// TIA Portal project "SistemaSemaforico_Curto_Claudio" (V15.1)

(* hardware
DEVICE "S7-1200 station_1"  S7-1200 Station
   slot 0: "Telaio di montaggio_0"  S7-1200 Rack  Rack  V1.0
   slot 1: "PLC_1"  CPU 1214C DC/DC/DC  6ES7 214-1AG40-0XB0  V4.2
*)

// ===== PLC "PLC_1"  CPU 1214C DC/DC/DC =====

VAR_GLOBAL   // PLC tag table "Tabella delle variabili standard"
   "Mutex" AT %M0.0 : Bool;
   "P" AT %I0.0 : Bool;
   "V1" AT %Q0.0 : Bool;
   "G1" AT %Q0.1 : Bool;
   "R1" AT %Q0.2 : Bool;
   "V2" AT %Q0.3 : Bool;
   "G2" AT %Q0.4 : Bool;
   "R2" AT %Q0.5 : Bool;
   "Abilita" AT %I0.1 : Bool;
   "Ped" AT %M0.1 : Bool;
END_VAR

VAR_GLOBAL CONSTANT   // PLC tag table "Tabella delle variabili standard"
   "Tempo_V" : Time := T#55s;
   "Tempo_R" : Time := T#60s;
   "Tempo_G" : Time := T#5s;
END_VAR

TYPE "VariabiliStato"
   STRUCT
      Home : Bool := true;
      Verde : Bool;
      Giallo : Bool;
      Rosso : Bool;
   END_STRUCT;
END_TYPE

DATA_BLOCK "Semaforo_DB"   // DB2
{ S7_Optimized_Access := 'TRUE' }
VERSION : 0.1
// stored: InstanceOfName Semaforo
"Semaforo"
BEGIN
END_DATA_BLOCK

DATA_BLOCK "Semaforo_DB_1"   // DB3
{ S7_Optimized_Access := 'TRUE' }
VERSION : 0.1
// stored: InstanceOfName Semaforo
"Semaforo"
BEGIN
END_DATA_BLOCK

// folder: System blocks/Program resources

DATA_BLOCK "IEC_Timer_0_DB"   // DB1
{ S7_Optimized_Access := 'TRUE' }
AUTHOR : Simatic
FAMILY : IEC
NAME : IEC_TMR
VERSION : 1.0
// stored: InstanceOfName IEC_TIMER
"IEC_TIMER"
BEGIN
END_DATA_BLOCK

// folder: (top level)

FUNCTION_BLOCK "Semaforo"   // FB1, LAD
{ S7_Optimized_Access := 'TRUE' }
VERSION : 0.1
   VAR_INPUT
      abilita : Bool;
   END_VAR
   VAR_OUTPUT
      V : Bool;
      G : Bool;
      R : Bool;
   END_VAR
   VAR_IN_OUT
      Mutex : Bool;
   END_VAR
   VAR RETAIN
      Stati : "VariabiliStato";
   END_VAR
   VAR_TEMP   // added for the SCL form of the ladder/FBD networks
      _w1 : Bool;
   END_VAR
BEGIN

REGION Network 1
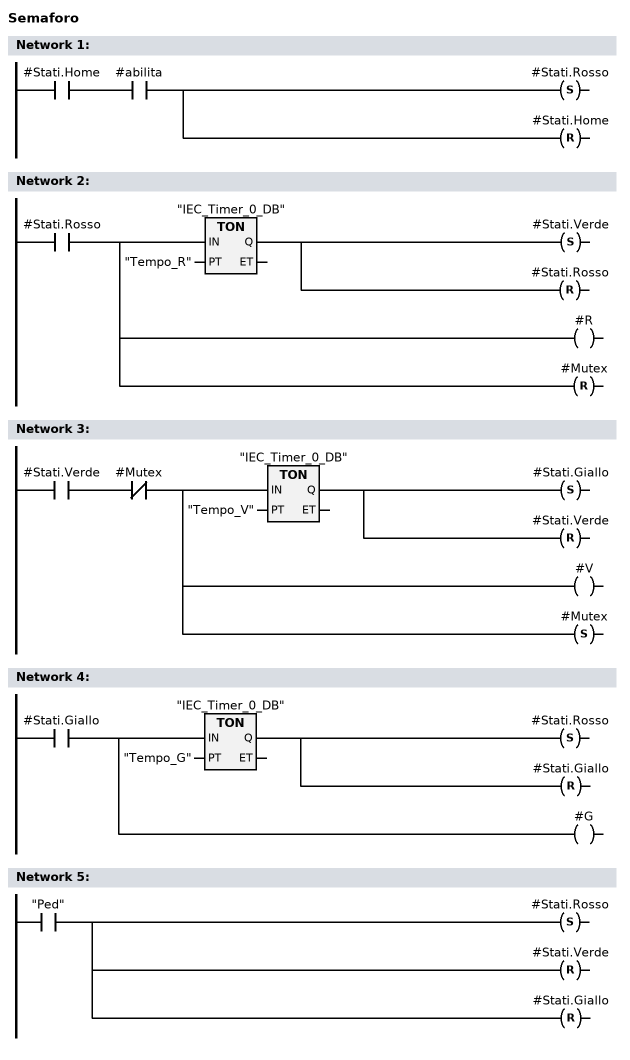
   RUNG wire#powerrail
      Contact( #Stati.Home )
      Contact( #abilita )
      wire#w1
      S_Coil( #Stati.Rosso )
   END_RUNG
   RUNG wire#w1
      R_Coil( #Stati.Home )
   END_RUNG
   // the same network as SCL:
   IF #Stati.Home AND #abilita THEN
       #Stati.Rosso := TRUE;
       #Stati.Home := FALSE;
   END_IF;
END_REGION

REGION Network 2
   "IEC_Timer_0_DB".TON(IN := #Stati.Rosso, PT := "Tempo_R");
   IF "IEC_Timer_0_DB".Q THEN #Stati.Verde := TRUE; END_IF;
   #_w1 := #Stati.Rosso;
   IF "IEC_Timer_0_DB".Q THEN #Stati.Rosso := FALSE; END_IF;
   #R := #_w1;
   IF #_w1 THEN #Mutex := FALSE; END_IF;
END_REGION

REGION Network 3
   #_w1 := #Stati.Verde AND NOT #Mutex;
   "IEC_Timer_0_DB".TON(IN := #_w1, PT := "Tempo_V");
   IF "IEC_Timer_0_DB".Q THEN
       #Stati.Giallo := TRUE;
       #Stati.Verde := FALSE;
   END_IF;
   #V := #_w1;
   IF #_w1 THEN #Mutex := TRUE; END_IF;
END_REGION

REGION Network 4
   "IEC_Timer_0_DB".TON(IN := #Stati.Giallo, PT := "Tempo_G");
   IF "IEC_Timer_0_DB".Q THEN #Stati.Rosso := TRUE; END_IF;
   #_w1 := #Stati.Giallo;
   IF "IEC_Timer_0_DB".Q THEN #Stati.Giallo := FALSE; END_IF;
   #G := #_w1;
END_REGION

REGION Network 5
   RUNG wire#powerrail
      Contact( "Ped" )
      wire#w1
      S_Coil( #Stati.Rosso )
   END_RUNG
   RUNG wire#w1
      R_Coil( #Stati.Verde )
   END_RUNG
   RUNG wire#w1
      R_Coil( #Stati.Giallo )
   END_RUNG
   // the same network as SCL:
   IF "Ped" THEN
       #Stati.Rosso := TRUE;
       #Stati.Verde := FALSE;
       #Stati.Giallo := FALSE;
   END_IF;
END_REGION
END_FUNCTION_BLOCK

ORGANIZATION_BLOCK "Main"   // OB1, LAD, ProgramCycle
TITLE = "Main Program Sweep (Cycle)"
{ S7_Optimized_Access := 'TRUE' }
VERSION : 0.1
   VAR_INPUT
      Initial_Call : Bool;   // Initial call of this OB
      Remanence : Bool;   // =True, if remanent data are available
   END_VAR
BEGIN

REGION Network 1
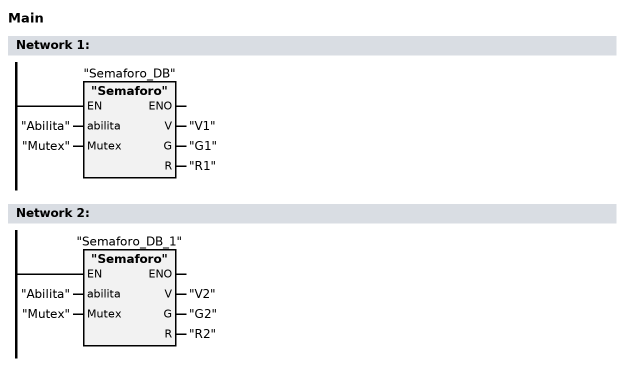
   RUNG wire#powerrail
      "Semaforo_DB"(abilita := "Abilita", Mutex := "Mutex", V => "V1", G => "G1", R => "R1")
   END_RUNG
   // the same network as SCL:
   "Semaforo_DB"(abilita := "Abilita", Mutex := "Mutex", V => "V1", G => "G1", R => "R1");   // "Semaforo"
END_REGION

REGION Network 2
   RUNG wire#powerrail
      "Semaforo_DB_1"(abilita := "Abilita", Mutex := "Mutex", V => "V2", G => "G2", R => "R2")
   END_RUNG
   // the same network as SCL:
   "Semaforo_DB_1"(abilita := "Abilita", Mutex := "Mutex", V => "V2", G => "G2", R => "R2");   // "Semaforo"
END_REGION
END_ORGANIZATION_BLOCK

ORGANIZATION_BLOCK "Pedone"   // OB40, LAD, HWProcessInterrupt
{ S7_Optimized_Access := 'TRUE' }
VERSION : 0.1
   VAR_INPUT
      LADDR : Hw_Io;   // Hardware identifier
      USI : Word;   // User structure identifier
      IChannel : USInt;   // Interrupt channel number
      EventType : Byte;   // EventType
   END_VAR
BEGIN

REGION Network 1
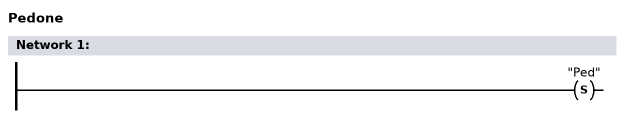
   RUNG wire#powerrail
      S_Coil( "Ped" )
   END_RUNG
   // the same network as SCL:
   "Ped" := TRUE;
END_REGION
END_ORGANIZATION_BLOCK